(* Schneider Machine Expert - Basic project TEST CUTBEND, file version 2.6.0.0 *)
(* ProjectInformations: Name=New project *)

HARDWARE
  Cpu 0: TM221CE40R
  EthernetConfiguration: NetworkName=M221, IpAllocationMode=FixedAddress, IpAddress=192.168.0.2, SubnetMask=255.255.255.0
  SerialLineConfiguration: Baud=Baud19200, Parity=ParityEven, DataBits=DataBits8, StopBits=StopBits1, PhysicalMedium=PhysicalMediumRs485, TransmissionMode=TransmissionModeModbusRtu, SlaveId=1, Addressing=SlaveAddressing
  MastTask: UsePeriodScanMode=false, PeriodScan=100
  FastTask: Period=255
  CpuBehavior: StartingMode=StartAsPreviousState, AutoSaveRamOnEeprom=true, WatchdogPeriod=250

SYMBOLS  (address, symbol, comment, settings)
  %M0         "START"
  %M1         "MOVE_TRF"
  %M2         "GRIPPER_C_CLOSE"
  %M3         "MOVE_BACK_TRF"
  %M4         "GRIPPER_ROTATE_CLOSE"
  %M5         "STATUS CB ON"
  %M6         "RELEASE_C_GRIPPER"
  %M7         "POLARITY_ RESULT"
  %M8         "POLARITY_CHECK"
  %M9         "ROTATE_0"
  %M10        "REVERSE_ROTATION"
  %M11        "RESET"
  %M12        "MANUAL"
  %M13        "CB_LF"
  %M14        "CB_RT"
  %M15        "ACTIVE_BOWLFEEDER"
  %M22        "LF_CB"
  %M23        "M_Q1"
  %M24        "M_Q2"
  %M25        "M_Q3"
  %M26      MANUAL_GRIP_CLOSE  "M_Q4"
  %M27        "M_Q5"
  %M28        "M_Q6"
  %M30        "EMG_Memory"
  %M31        "Start_Memory"
  %M47        "M_EMG"
  %M49        "POLARITY CHECKED"
  %M50        "NEGATIVE"
  %M51        "POSITIVE"
  %M52        "FIRST RUN"
  %M53        "DONE CUTTING"
  %M54        "NEGATIVE READY"
  %M55        "TRIGGER"
  %M56        "COUNTER OUTPUT"
  %M100       "START GUI"
  %M102       "M_START"
  %MW0        "Count Output"
  %TM0        [Preset=1, Base=OneSecond]
  %TM1        [Preset=1, Base=OneSecond]
  %TM2        [Preset=1, Base=OneSecond]
  %I0.0       "EMG"
  %I0.1       "BTN START"
  %I0.2       "LF_CB_FWD"
  %I0.3       "LF_CB_BWD"
  %I0.4       "RT_CB_FWD"
  %I0.5       "RT_CB_BWD"
  %I0.6       "R_CW"
  %I0.7       "R_CCW"
  %I0.8       "GRIP_R_OPEN"
  %I0.9       "GRIP_R_CLOSE"
  %I0.10      "GRIP_C_OPEN"
  %I0.11      "GRIP_C_CLOSE"
  %I0.12      "C_TRF_FWD"
  %I0.13      "C_TRF_FWD"
  %I0.14      "PART_DETECTION"
  %I0.15      "POLARITY"
  %Q0.0       "LF_CB"
  %Q0.1       "RT_CB"
  %Q0.2       "R_P"
  %Q0.3       "GRIP_COMP"
  %Q0.4       "GRIP_ROTATE"
  %Q0.5       "TRF_C"
  %Q0.6       "BOWL_FEEDER"

POU Bowl Feeder
  (* SectionNumber=1 *)

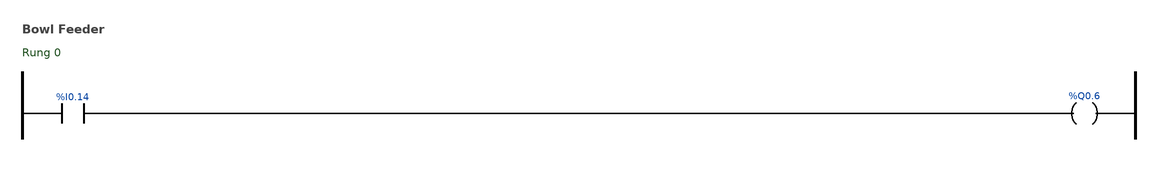

// Rung 0
  LD %I0.14
  ST %Q0.6
  // as ST:
  //   %Q0.6 := %I0.14;

POU START
  (* SectionNumber=2 *)

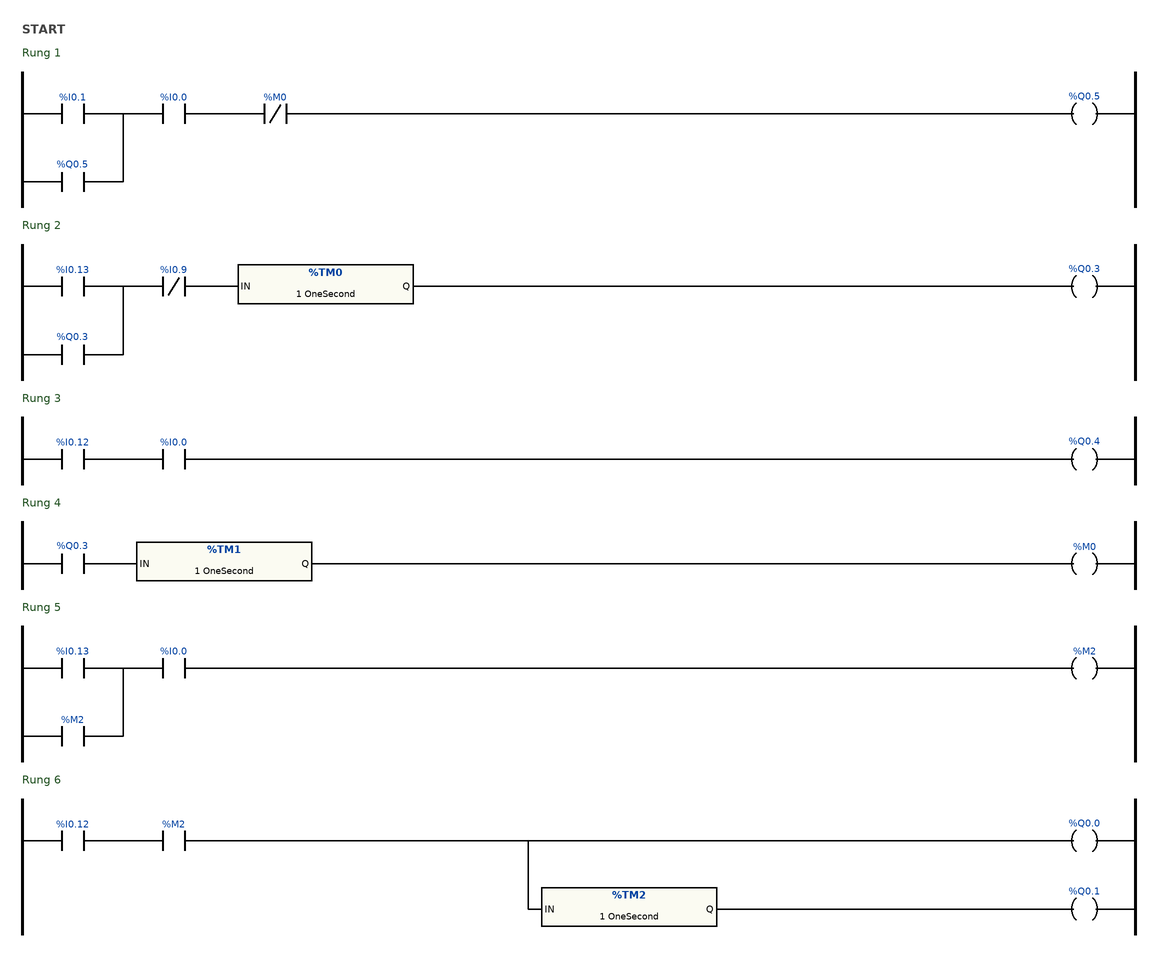

// Rung 1
  LD %I0.1
  OR %Q0.5
  AND %I0.0
  ANDN %M0
  ST %Q0.5
  // as ST:
  //   %Q0.5 := (%I0.1 OR %Q0.5) AND %I0.0 AND NOT %M0;

// Rung 2
  BLK %TM0
  LD %I0.13
  OR %Q0.3
  ANDN %I0.9
  IN
  OUT_BLK
  LD Q
  ST %Q0.3
  END_BLK
  // as ST:
  //   %TM0(IN := (%I0.13 OR %Q0.3) AND NOT %I0.9);
  //   %Q0.3 := %TM0.Q;

// Rung 3
  LD %I0.12
  AND %I0.0
  ST %Q0.4
  // as ST:
  //   %Q0.4 := %I0.12 AND %I0.0;

// Rung 4
  BLK %TM1
  LD %Q0.3
  IN
  OUT_BLK
  LD Q
  ST %M0
  END_BLK
  // as ST:
  //   %TM1(IN := %Q0.3);
  //   %M0 := %TM1.Q;

// Rung 5
  LD %I0.13
  OR %M2
  AND %I0.0
  ST %M2
  // as ST:
  //   %M2 := (%I0.13 OR %M2) AND %I0.0;

// Rung 6
  LD 1
  MULTIFB
  LD 1
  AND %I0.12
  AND %M2
  ST %MW2009:X0
  LD %MW2009:X0
  ST %Q0.0
  BLK %TM2
  LD %MW2009:X0
  IN
  OUT_BLK
  LD Q
  ST %Q0.1
  END_BLK
  MULTIFB
  // as ST:
  //   %Q0.0 := %I0.12 AND %M2;
  //   %TM2(IN := %I0.12 AND %M2);
  //   %Q0.1 := %TM2.Q;
